FUNCTION IsReady : BOOL
VAR_INPUT
	Condition : BOOL;
END_VAR

IsReady := Condition;

END_FUNCTION

(* stored: Version 1.1.0.1, ProductVersion 3.1.4024.15
   POU IsReady: Id {0aac700e-f7ce-44e5-beb3-86f2d77b0971}, SpecialFunc None *)
